{attribute wpf [Container(Layout.Wrap)]}
TYPE WrapLayoutTest :
STRUCT
	test1: BOOL;
	var1: INT;
	test2: STRING;
	
	
	simulation : RealValueSimulation;
END_STRUCT
END_TYPE

(* stored: Version 1.1.0.1, ProductVersion 3.1.4024.9
   DUT WrapLayoutTest: Id {3889ad76-98dd-498a-bef0-7ecba1d20f63} *)
